FUNCTION_BLOCK CardboardCornerGuardEx EXTENDS SectionEx
VAR
	robotLeft, robotRight : REFERENCE TO Robot;
	
	insertionLeft, insertionRight : REFERENCE TO Insertion;
	insertionBottom : REFERENCE TO TeknicEIP;
	
	wrapper : REFERENCE TO WrapMachine;
	overhead : REFERENCE TO STRING;
	
	skidLeft, skidRight : REFERENCE TO MaterialStorage; //cardboard
	magazineLeft, magazineRight : REFERENCE TO MaterialStorage; //corner guard
	
	benderLeft : REFERENCE TO FoldingMachine;
END_VAR
VAR
	pushConveyorPos: REAL;
	wrapConveyorPos : REAL;
	
	insertionSlots : ARRAY[Surface.TOP_LEFT..Surface.BOTTOM_RIGHT] OF STRING;
	
	combinedCardboardCornerGuard : ARRAY[0..2*GVL.maxPairs] OF PositionMaterials;
	recipesCombined : BOOL;
	
	materialsArr : POINTER TO PositionMaterials; //array of PositionMaterials
	currentPair : REFERENCE TO PositionMaterials;
	
	frontCoverPlaced : BOOL;
	backCoverPlaced : BOOL;
	
	cornerSetLeft, cornerSetRight : INT;
	
	iWrap : INT;
	
	step : (PLACE_FRONT_COVER := -10, PLACE_BACK_COVER := -20, RUN_TO_POSITION, LOAD_FLATS, PUSH, RUN_TO_WRAP_POSITION, WRAP_AND_RELEASE, RESET);
	robotLeftOutputs, robotRightOutputs : ARRAY[1..50] OF INT;
END_VAR

entryRefPos := pushConveyorPos;
exitRefPos := wrapConveyorPos;

SUPER^();

CASE status OF
	SectionStatus.IDLE:
		RETURN;
	
	SectionStatus.ALIGNING:
		IF NOT recipesCombined THEN
			combine(
				currentBundle.cardboard, 
				currentBundle.cornerGuard, 
				combinedCardboardCornerGuard, 
				currentBundle.cardboard_over_cornerGuard);
				
			recipesCombined := TRUE;
		END_IF
		
	SectionStatus.ACTIVE:
		recipesCombined := FALSE;
		
	SectionStatus.CLEARING:
		//
		
	SectionStatus.COMPLETE:	
		//
		
	-100:
		RETURN;
		
END_CASE

METHOD changeRobotsEOAT : BOOL
VAR_INPUT
END_VAR
(*
IF robotLeft.tool <> sectionID THEN
	MEMSET(ADR(robotLeftOutputs), 0, SIZEOF(robotLeftOutputs));
	//robotLeftOutputs[1] := A21.TOOL_CHANGE_CHIPBOARD;
	robotLeft.setParamsAndWait(robotLeftOutputs);
END_IF

IF robotRight.tool <> sectionID THEN
	MEMSET(ADR(robotRightOutputs), 0, SIZEOF(robotRightOutputs));
	//robotRightOutputs[1] := A21.TOOL_CHANGE_CHIPBOARD;
	robotRight.setParamsAndWait(robotRightOutputs);
END_IF

changeRobotsEOAT := robotLeft.tool = sectionID AND robotRight.tool = sectionID;
*)
END_METHOD

METHOD PROTECTED combine : BOOL
VAR_IN_OUT
	cardboard : ARRAY[*] OF PositionMaterials;
	cornerGuard : ARRAY[*] OF PositionMaterials;
	
	combined : ARRAY[*] OF PositionMaterials;
END_VAR
VAR_INPUT
	cardboard_over_cornerGuard : BOOL;
END_VAR
VAR_INST
	topLength : REAL;
	leftLength : REAL;
	rightLength : REAL;
	bottomLength : REAL;
	
	topLeftLength : REAL;
	topRightLength : REAL;
	bottomLeftLength : REAL;
	bottomRightLength : REAL;
	
	outerMaterialLength : REAL;
	innerMaterialLength : REAL;
	
	i : INT;
	iCardboard : INT;
	iCornerGuard : INT;
END_VAR
FOR i:=0 TO GVL.maxPairs*2 BY 1 DO
	IF //no more cardboard (reached end of array or unused entries), 
		(iCardboard >= GVL.maxPairs OR_ELSE NOT PositionIsValid(cardboard[iCardboard])) AND_THEN //no more valid cardboard entries
		iCornerGuard < GVL.maxPairs AND_THEN //still has remaining corner guard
		PositionIsValid(cornerGuard[iCornerGuard]) //remaining corner guard is valid		
	THEN //finish with cornerguard
		combined[i] := cornerGuard[iCornerGuard];
		iCornerGuard := iCornerGuard + 1;
		CONTINUE;
	END_IF
	
	IF //no more cornerguard (reached end of array or unused entries)
		(iCornerGuard >= GVL.maxPairs OR_ELSE NOT PositionIsValid(cornerGuard[iCornerGuard])) AND_THEN
		iCardboard < GVL.maxPairs AND_THEN
		PositionIsValid(cardboard[iCardboard])
	THEN //finish with cardboard
		combined[i] := cardboard[iCardboard];
		iCardboard := iCardboard + 1;
		CONTINUE;
	END_IF
	
	(*
	IF NOT cardboard_over_cornerGuard THEN //cardboard on inside
		setOrder(cardboard, cornerGuard, combined, iCardboard, iCornerGuard, i);
		
	ELSE //cardboard on outside
		setOrder(cornerGuard, cardboard, combined, iCornerGuard, iCardboard, i);
		
	END_IF
	*)
END_FOR

combine := TRUE;
END_METHOD

METHOD initHardware : BOOL
conveyors := ADR(allConveyors);

robotLeft REF= robots[3];
robotRight REF= robots[4];
(*
insertionLeft REF= Hardware.insertionCardboardCornerGuardSides[Surface.LEFT];
insertionRight REF= Hardware.insertionCardboardCornerGuardSides[Surface.RIGHT];

wrapper REF= Hardware.wrapperCardboardCornerguard;
overhead REF= Hardware.overhead;

skidLeft REF= Hardware.cardboardSkid[Surface.LEFT];
skidRight REF= Hardware.cardboardSkid[Surface.RIGHT];

magazineLeft REF= Hardware.cornerGuardMagazine[Surface.LEFT];
magazineRight REF= Hardware.cornerGuardMagazine[Surface.RIGHT];

benderLeft REF= Hardware.cardboardBender[Surface.LEFT];
*)

insertionLeft REF= insertionA22Left;
insertionRight REF= insertionA22Right;

wrapper REF= wrapperA22;
overhead REF= Hardware.overhead;

skidLeft REF= cardboardSkidLeft;
skidRight REF= cardboardSkidRight;

magazineLeft REF= cornerGuardMagazineLeft;
magazineRight REF= cornerGuardMagazineRight;

benderLeft REF= cardboardBenderLeft;
END_METHOD

METHOD PROTECTED leftBendingSequence : BOOL
VAR_IN_OUT
	actingRobot : Robot;
	actingSkid : MaterialStorage;
	
	actingLoadStep : INT;
	actingRobotStep : INT;
END_VAR
VAR_INPUT
	materialID : STRING;
	foldPosition1 : INT;
	foldPosition2 : INT;
END_VAR
VAR_OUTPUT
	fail : BOOL;
END_VAR
VAR
	slot : INT;
END_VAR
END_METHOD

METHOD PROTECTED leftOverheadSequence : BOOL
VAR_IN_OUT
	actingRobot : Robot;
	actingSkid : MaterialStorage;
	
	actingLoadStep : INT;
	actingRobotStep : INT;
END_VAR
VAR_INPUT
	materialID : STRING;
	foldPosition1 : INT;
	foldPosition2 : INT;
END_VAR
VAR_OUTPUT
	fail : BOOL;
END_VAR
VAR
	slot : INT;
END_VAR
(*
CASE actingLoadStep OF
	0: //skid to bender
		IF NOT actingSkid.findSlot(materialID, position=> slot) THEN
			fail := TRUE;
			RETURN;
		END_IF
		
		IF
			actingRobot.reserve() AND_THEN
			actingRobot.setCommandAndWait(
				task:= A22.TRANSFER_TO_BENDER, 
				param0:= slot, 
				param1:= foldPosition1, 
				param2:= foldPosition2)
		THEN
			actingRobotStep := 10;
		END_IF
		
	10: //bend
		(*
		IF bendingMachine.done THEN
			cardboardCornersLoadStep := 20;
		END_IF
		*)
		
	20: //bender to overhead
		IF overhead <> '' THEN
			RETURN;
		END_IF
		
		IF
			actingRobot.reserve() AND_THEN
			actingRobot.setCommandAndWait(
				task:= A22.TRANSFER_TO_OVERHEAD, 
				param0:= 0, 
				param1:= 0, 
				param2:= 0)
		THEN
			actingRobotStep := 10;
		END_IF
		
		CASE actingRobotStep OF
			COMMAND: //send command
				IF NOT actingRobot.reserve() THEN
					RETURN;
				END_IF
				
				IF actingSkid.findSlot(currentPair.topRight, position=> slot) THEN
					actingRobot.command(
						task:= A22.TRANSFER_TO_OVERHEAD, 
						param0:= 0, 
						param1:= 0, 
						param2:= 0);
						
				ELSE
					fail := TRUE;
					RETURN;
					
				END_IF
				
			WAIT:
				IF actingRobot.done THEN
					overhead := materialID;
					
					actingRobot.release();
					actingRobotStep := 30;
					actingLoadStep := Surface.BOTTOM_RIGHT;
				END_IF
		END_CASE
END_CASE
*)
END_METHOD

METHOD PROTECTED leftRobotCornersSequence : BOOL
VAR_IN_OUT
	actingRobot : Robot;
	skid : MaterialStorage;
	loadStep : INT;
END_VAR
VAR_INPUT
	surfaceID : Surface;
	materialID : STRING;
	foldPos0 : INT;
	foldPos1 : INT;
END_VAR
VAR_OUTPUT
	fail : BOOL;
END_VAR
VAR
	slot : INT;
	
	task : INT;
	param0, param1, param2 : INT;
END_VAR
IF materialID = '' THEN
	leftRobotCornersSequence := TRUE;
	RETURN;
END_IF

IF NOT benderLeft.busy THEN
	benderLeft.foldPos0 := foldPos0;
	benderLeft.foldPos1 := foldPos1;
END_IF

CASE loadStep OF
	0: //skid to bender
		IF NOT skid.findSlot(materialID, atSlot=> slot) THEN
			fail := TRUE;
			RETURN;
		END_IF
		
		IF
			actingRobot.setCommandAndWait(
				task:= A22.TRANSFER_TO_BENDER, 
				param1:= slot, 
				param2:= foldPos0, 
				param3:= foldPos1)
		THEN
			loadStep := 10;
		END_IF
		
	10: //bend
		//IF benderLeft.done THEN
			loadStep := 20;
		//END_IF
		
		
	20: //bender to overhead or left insertion
		CASE surfaceID OF
			Surface.TOP_RIGHT, Surface.BOTTOM_RIGHT: //transfer to overhead
				IF overhead <> '' THEN
					RETURN;
				END_IF
				task := A22.TRANSFER_TO_OVERHEAD;
				
			Surface.TOP_LEFT: //load to insertion
				task:= A22.LOAD_BENDER_TO_UPPER_CORNER;
					
			Surface.BOTTOM_LEFT: //load to insertion
				task := A22.LOAD_BENDER_TO_LOWER_CORNER;
				
		END_CASE
		
		IF
			actingRobot.setCommandAndWait(
				task:= task, 
				param1:= param0, 
				param2:= param1, 
				param3:= param1)
		THEN
			 loadStep := COMPLETE;
		END_IF
	
	COMPLETE:
		//turn on suction
		leftRobotCornersSequence := TRUE;
	
END_CASE
END_METHOD

METHOD PROTECTED load : BOOL
VAR_INPUT
	pair : REFERENCE TO PositionMaterials;
END_VAR
VAR
	nextPair : REFERENCE TO PositionMaterials REF= materialsArr[iPair + 1];
	finished : BOOL;
END_VAR
(*
this method only loads corner materials (L-cardboards and corner guards)
to load flat cardboards, use loadFlats()
*)

IF NOT (robotLeft.operational AND robotRight.operational) THEN
	error := TRUE;
	currentBypass := TRUE;
	RETURN;
END_IF

IF NOT (robotLeft.reserve(sectionID) AND robotRight.reserve(sectionID)) THEN //both robots must be reserved first
	RETURN;
END_IF


IF //if next material has same position as this material, only happens if this material is cardboard and next is corner guard
	nextPair.position = pair.position AND_THEN
	NOT loadCornerGuards(nextPair, fail=> ) //load next pair (corner guards) first
THEN
	RETURN;
END_IF


IF MatchesMaterialType(pair:= pair, materialType:= 'CAR') THEN //is cardboard
	load := loadCornerCardboards(pair:= pair);

ELSIF MatchesMaterialType(pair:= pair, materialType:= 'COR') THEN //is corner guard
	load := loadCornerGuards(pair:= pair);

END_IF


IF load THEN
	robotLeft.release(sectionID);
	robotRight.release(sectionID);
END_IF
END_METHOD

METHOD PROTECTED loadBottom : BOOL
VAR_IN_OUT
	actingRobot : Robot;
	actingStorage : MaterialStorage;
	actingLoadStep : INT;
END_VAR
VAR_INPUT
	material : STRING;
END_VAR
VAR_OUTPUT
	fail : BOOL;
END_VAR
VAR
	slot : INT;
END_VAR
IF material = '' THEN
	loadBottom := TRUE;
	RETURN;
END_IF

CASE actingLoadStep OF
	0:
		IF NOT actingStorage.findSlot(materialID := material, atSlot => slot) THEN
			fail := TRUE;
			RETURN;
		END_IF
		
		IF
			actingRobot.setCommandAndWait( //perform the task
				task:= A22.LOAD_CARDBOARD_BOTTOM,
				param1:= slot,
				param2:= 0,
				param3:= 0)
		THEN
			actingLoadStep := COMPLETE;
		END_IF
		
	COMPLETE:
		//turn on suction
		loadBottom := TRUE;
	
END_CASE
END_METHOD

METHOD PROTECTED loadBottomLeft : BOOL
VAR_IN_OUT
	actingRobot : Robot;
	actingStorage : MaterialStorage;
	actingLoadStep : INT;
END_VAR
VAR_INPUT
	material : STRING;
END_VAR
VAR_OUTPUT
	fail : BOOL;
END_VAR
VAR
	slot : INT;
END_VAR
IF material = '' THEN
	loadBottomLeft := TRUE;
	RETURN;
END_IF

CASE actingLoadStep OF
	0:
		IF NOT actingStorage.findSlot(materialID := material, atSlot => slot) THEN //load from staging table
			fail := TRUE;
			RETURN;
		END_IF
		
		IF
			actingRobot.setCommandAndWait( //perform the task
				task:= A22.LOAD_CORNER_GUARD_LOWER,
				param1:= slot,
				param2:= 0,
				param3:= 0)
		THEN
			actingLoadStep := COMPLETE;
		END_IF
		
	COMPLETE:
		loadBottomLeft := TRUE;
END_CASE
END_METHOD

METHOD PROTECTED loadBottomRight : BOOL
VAR_IN_OUT
	actingRobot : Robot;
	actingStorage : MaterialStorage;
	actingLoadStep : INT;
END_VAR
VAR_INPUT
	material : STRING;
END_VAR
VAR_OUTPUT
	fail : BOOL;
END_VAR
VAR
	slot : INT;
END_VAR
IF material = '' THEN
	loadBottomRight := TRUE;
	RETURN;
END_IF

CASE actingLoadStep OF
	0:
		IF NOT actingStorage.findSlot(materialID := material, atSlot => slot) THEN //load from staging table
			fail := TRUE;
			RETURN;
		END_IF
		
		IF
			actingRobot.setCommandAndWait( //perform the task
				task:= A22.LOAD_CORNER_GUARD_LOWER,
				param1:= slot,
				param2:= 0,
				param3:= 0)
		THEN
			actingLoadStep := COMPLETE;
		END_IF
		
	COMPLETE:
		loadBottomRight := TRUE;
END_CASE
END_METHOD

METHOD PROTECTED loadCornerCardboards : BOOL
VAR_INPUT
	pair : REFERENCE TO PositionMaterials;
END_VAR
IF cornerSetLeft = 0 THEN //LEFT SIDE
	cornerSetLeft := Surface.TOP_RIGHT;
END_IF

IF
	leftRobotCornersSequence(
		actingRobot:= robotLeft, 
		skid:= skidLeft, 
		surfaceID:= cornerSetLeft,
		loadStep:= loadStepLeft, 
		materialID:= pair.topRight, 
		foldPos0:= currentBundle.cardboardFolds[cornerSetLeft][iPair],
		foldPos1:= 0,
		fail=> )
THEN
	CASE cornerSetLeft OF
		Surface.TOP_RIGHT: 
			cornerSetLeft := Surface.TOP_LEFT;
			loadStepLeft := 0;
			
		Surface.TOP_LEFT: 
			cornerSetLeft := Surface.BOTTOM_RIGHT;
			loadStepLeft := 0;
			
		Surface.BOTTOM_RIGHT: 
			cornerSetLeft := Surface.BOTTOM_LEFT;
			loadStepLeft := 0;
			
		Surface.BOTTOM_LEFT: 
			cornerSetLeft := COMPLETE;
			loadStepLeft := COMPLETE;
			
		COMPLETE:
			//
			
	END_CASE
END_IF



IF cornerSetRight = 0 THEN //RIGHT SIDE
	cornerSetRight := Surface.TOP_RIGHT;
END_IF

IF
	rightRobotCornersSequence(
		actingRobot:= robotRight, 
		skid:= skidRight, 
		loadStep:= loadStepRight, 
		materialID:= pair.topRight, 
		surfaceID:= cornerSetRight,
		foldPos1:= currentBundle.cardboardFolds[cornerSetRight][iPair], 
		foldPos2:= 0, 
		fail=> )
THEN
	CASE cornerSetRight OF
		Surface.TOP_RIGHT: 
			cornerSetRight := Surface.BOTTOM_RIGHT;
			loadStepRight := 0;
			
		Surface.BOTTOM_RIGHT: 
			cornerSetRight := COMPLETE;			
			loadStepRight := COMPLETE;
			
		COMPLETE:
			//
			
	END_CASE
END_IF


IF cornerSetLeft = COMPLETE AND cornerSetRight = COMPLETE THEN
	loadCornerCardboards := TRUE;
	
	loadStepLeft := loadStepRight := 0;
	cornerSetLeft := cornerSetRight := 0;
END_IF
END_METHOD

METHOD PROTECTED loadCornerGuards : BOOL
VAR_INPUT
	pair : REFERENCE TO PositionMaterials;
END_VAR
VAR_OUTPUT
	fail : BOOL;
END_VAR
VAR
	leftFail : BOOL;
	rightFail : BOOL;
END_VAR
CASE loadSet OF
	0: //upper corners
		IF 
			loadCornerGuardSequence(
				actingRobot:= robotLeft, 
				robotOutputs:= robotLeftOutputs, 
				actingStorage:= skidLeft, 
				actingLoadStep:= loadStepLeft, 
				surfaceID:= Surface.TOP_LEFT, 
				material:= pair.topLeft, 
				fail=> leftFail)
			AND
			loadCornerGuardSequence(
				actingRobot:= robotRight, 
				robotOutputs:= robotRightOutputs, 
				actingStorage:= skidRight,
				actingLoadStep:= loadStepRight, 
				surfaceID:= Surface.TOP_RIGHT, 
				material:= pair.topRight, 
				fail=> rightFail)
		THEN
			loadStepLeft := loadStepRight := 0;
			loadSet := 10;
		END_IF
		
	10: //lower corners
		IF 
			loadCornerGuardSequence(
				actingRobot:= robotLeft, 
				robotOutputs:= robotLeftOutputs, 
				actingStorage:= skidLeft, 
				actingLoadStep:= loadStepLeft, 
				surfaceID:= Surface.BOTTOM_LEFT, 
				material:= pair.bottomLeft, 
				fail=> leftFail)
			AND
			loadCornerGuardSequence(
				actingRobot:= robotRight, 
				robotOutputs:= robotRightOutputs, 
				actingStorage:= skidRight,
				actingLoadStep:= loadStepRight, 
				surfaceID:= Surface.BOTTOM_RIGHT, 
				material:= pair.bottomRight, 
				fail=> rightFail)
		THEN
			loadStepLeft := loadStepRight := 0;
			loadSet := COMPLETE;
		END_IF
	
	COMPLETE:
		loadStepLeft := loadStepRight := 0;
		loadSet := 0;
		
		loadCornerGuards := TRUE;
END_CASE

fail := MAX(leftFail, rightFail);
END_METHOD

METHOD loadCornerGuardSequence : BOOL
VAR_IN_OUT
	actingRobot : Robot;
	robotOutputs : ARRAY[1..50] OF INT;
	actingStorage : MaterialStorage;
	actingLoadStep : INT;
END_VAR
VAR_INPUT
	surfaceID : Surface;
	material : STRING;
END_VAR
VAR_OUTPUT
	fail : BOOL;
END_VAR
VAR
	slot : INT;
END_VAR
IF material = '' THEN
	loadCornerGuardSequence := TRUE;
	RETURN;
END_IF

CASE actingLoadStep OF
	0:
		IF NOT actingStorage.findSlot(materialID := material, atSlot => slot) THEN //load from staging table
			fail := TRUE;
			RETURN;
		END_IF
		
		MEMSET(ADR(robotOutputs), 0, SIZEOF(robotOutputs));
		CASE surfaceID OF
			Surface.TOP_LEFT, Surface.TOP_RIGHT: 		robotOutputs[1] := A22.LOAD_CORNER_GUARD_UPPER;
			Surface.BOTTOM_LEFT, Surface.BOTTOM_RIGHT:	robotOutputs[1] := A22.LOAD_CORNER_GUARD_LOWER;
		END_CASE
		robotOutputs[2] := slot;
		
		IF actingRobot.setParamsAndWait(robotOutputs) THEN
			actingLoadStep := COMPLETE;
		END_IF
		
	COMPLETE:
		//outerSuctions[surfaceID].enable := TRUE;
		loadCornerGuardSequence := TRUE;
END_CASE
END_METHOD

METHOD PROTECTED loadFlats : BOOL
VAR_INPUT
	pair : REFERENCE TO PositionMaterials;
END_VAR
CASE loadSet OF
	0: //top and bottom
		IF 
			loadTop(robotLeft, skidLeft, loadStepLeft, pair.top, fail=> ) AND
			loadBottom(robotRight, skidRight, loadStepRight, pair.bottom, fail=> )
		THEN
			loadStepLeft := loadStepRight := 0;
			loadSet := 10;
		END_IF
		
	10: //sides
		IF 
			loadSides(robotLeft, skidLeft, loadStepLeft, pair.top, fail=> ) AND
			loadSides(robotRight, skidRight, loadStepRight, pair.bottom, fail=> )
		THEN
			loadStepLeft := loadStepRight := 0;
			loadSet := COMPLETE;
		END_IF
	
	COMPLETE:
		loadStepLeft := loadStepRight := 0;
		loadSet := 0;
		
		loadFlats := TRUE;
END_CASE
END_METHOD

METHOD loadFlatSequence : BOOL
VAR_IN_OUT
	actingRobot : Robot;
	robotOutputs : ARRAY[1..50] OF INT;
	actingStorage : MaterialStorage;
	actingLoadStep : INT;
END_VAR
VAR_INPUT
	surfaceID : Surface;
	material : STRING;
END_VAR
VAR_OUTPUT
	fail : BOOL;
END_VAR
VAR
	slot : INT;
END_VAR
IF material = '' THEN
	loadFlatSequence := TRUE;
	RETURN;
END_IF

CASE actingLoadStep OF
	0:
		IF NOT actingStorage.findSlot(materialID := material, atSlot => slot) THEN
			fail := TRUE;
			RETURN;
		END_IF
		
		MEMSET(ADR(robotOutputs), 0, SIZEOF(robotOutputs));
		CASE surfaceID OF
			Surface.TOP: 					robotOutputs[1] := A22.LOAD_CARDBOARD_TOP;
			Surface.LEFT, Surface.RIGHT: 	robotOutputs[1] := A22.LOAD_CARDBOARD_SIDE;
			Surface.BOTTOM: 				robotOutputs[1] := A22.LOAD_CARDBOARD_BOTTOM;
		END_CASE
		robotOutputs[2] := slot;
		
		IF actingRobot.setParamsAndWait(robotOutputs) THEN
			actingLoadStep := COMPLETE;
		END_IF
		
	COMPLETE:
		loadFlatSequence := TRUE;
	
END_CASE
END_METHOD

METHOD PROTECTED loadSides : BOOL
VAR_IN_OUT
	actingRobot : Robot;
	actingStorage : MaterialStorage;
	actingLoadStep : INT;
END_VAR
VAR_INPUT
	material : STRING;
END_VAR
VAR_OUTPUT
	fail : BOOL;
END_VAR
VAR
	slot : INT;
END_VAR
IF material = '' THEN
	loadSides := TRUE;
	RETURN;
END_IF

CASE actingLoadStep OF
	0:
		IF NOT actingStorage.findSlot(materialID := material, atSlot => slot) THEN
			fail := TRUE;
			RETURN;
		END_IF
		
		IF
			actingRobot.setCommandAndWait( //perform the task
				task:= A22.LOAD_CARDBOARD_SIDE,
				param1:= slot,
				param2:= 0,
				param3:= 0)
		THEN
			actingLoadStep := COMPLETE;
		END_IF
		
	COMPLETE:
		//turn suction on
		loadSides := TRUE;
END_CASE
END_METHOD

METHOD PROTECTED loadTop : BOOL
VAR_IN_OUT
	actingRobot : Robot;
	actingStorage : MaterialStorage;
	actingLoadStep : INT;
END_VAR
VAR_INPUT
	material : STRING;
END_VAR
VAR_OUTPUT
	fail : BOOL;
END_VAR
VAR
	slot : INT;
END_VAR
IF material = '' THEN
	loadTop := TRUE;
	RETURN;
END_IF

CASE actingLoadStep OF
	0:
		IF NOT actingStorage.findSlot(materialID := material, atSlot => slot) THEN //load from staging table
			fail := TRUE;
			RETURN;
		END_IF
		
		IF
			actingRobot.setCommandAndWait( //perform the task
				task:= A22.LOAD_CARDBOARD_TOP,
				param1:= slot,
				param2:= 0,
				param3:= 0)
		THEN
			actingLoadStep := COMPLETE;
		END_IF
		
	COMPLETE:
		loadTop := TRUE;
END_CASE
END_METHOD

METHOD PROTECTED loadTopLeft : BOOL
VAR_IN_OUT
	actingRobot : Robot;
	actingStorage : MaterialStorage;
	actingLoadStep : INT;
END_VAR
VAR_INPUT
	material : STRING;
END_VAR
VAR_OUTPUT
	fail : BOOL;
END_VAR
VAR
	slot : INT;
END_VAR
IF material = '' THEN
	loadTopLeft := TRUE;
	RETURN;
END_IF

CASE actingLoadStep OF
	0:
		IF NOT actingStorage.findSlot(materialID := material, atSlot => slot) THEN //load from staging table
			fail := TRUE;
			RETURN;
		END_IF
		
		IF
			actingRobot.setCommandAndWait( //perform the task
				task:= A22.LOAD_CORNER_GUARD_UPPER,
				param1:= slot,
				param2:= 0,
				param3:= 0)
		THEN
			actingLoadStep := COMPLETE;
		END_IF
		
	COMPLETE:
		loadTopLeft := TRUE;
END_CASE
END_METHOD

METHOD PROTECTED loadTopRight : BOOL
VAR_IN_OUT
	actingRobot : Robot;
	actingStorage : MaterialStorage;
	actingLoadStep : INT;
END_VAR
VAR_INPUT
	material : STRING;
END_VAR
VAR_OUTPUT
	fail : BOOL;
END_VAR
VAR
	slot : INT;
END_VAR
IF material = '' THEN
	loadTopRight := TRUE;
	RETURN;
END_IF

CASE actingLoadStep OF
	0:
		IF NOT actingStorage.findSlot(materialID := material, atSlot => slot) THEN //load from staging table
			fail := TRUE;
			RETURN;
		END_IF
		
		IF
			actingRobot.setCommandAndWait( //perform the task
				task:= A22.LOAD_CORNER_GUARD_UPPER,
				param1:= slot,
				param2:= 0,
				param3:= 0)
		THEN
			actingLoadStep := COMPLETE;
		END_IF
		
	COMPLETE:
		loadTopRight := TRUE;
END_CASE
END_METHOD

METHOD placeFrontCover : BOOL
VAR_INPUT
END_VAR
END_METHOD

METHOD PROTECTED process : BOOL
VAR
	masterLength : REAL;
	targetPos : REAL;
	targetStep : INT;
END_VAR
VAR
	maxHeight : REAL := 1000; //1000mm, 100cm, 1m tall at home pos
END_VAR
(*
VAR_INST
	resumePosition : REAL;
END_VAR
VAR CONSTANT
	wrapDelta : REAL := 5;
END_VAR
*)
//TODO: write instructions for wrapping front and back covers

IF NOT frontCoverPlaced THEN
	targetPos := 0;
	
ELSIF iPair < GVL.maxPairs THEN
	targetPos := currentPair.position;
	
ELSIF NOT backCoverPlaced AND iPair >= GVL.maxPairs THEN
	targetPos := currentBundle.length;
	
ELSIF iPair >= GVL.maxPairs THEN
	process := TRUE;
	RETURN;
	
END_IF

CASE step OF
	PLACE_FRONT_COVER:
		IF placeFrontCover() THEN
			step := RUN_TO_POSITION;
		END_IF
	
	RUN_TO_POSITION:
		IF //only load corners, flats will be PUSHed when bundle arrives at position
			directionCheckAndSet(pushConveyorPos, currentPair.position) AND 
			load(pair:= currentPair)
		THEN
			step := 10;
		END_IF
		
	LOAD_FLATS:
		IF loadFlats(pair:= currentPair) THEN
			step := PUSH;
		END_IF
		
	PUSH:
		setConveyorMode(ConveyorMode.STOP);
		(*
		IF
			NOT insertionLeft.align(targetPos:= maxHeight - currentBundle.height) OR
			NOT insertionRight.align(targetPos:= maxHeight - currentBundle.height)
		THEN
			RETURN;
		END_IF
		
		insertionLeft.press();
		insertionRight.press();
		*)
		
		IF NOT insertionLeft.contact THEN
			//insertionRight.slideOut();
			insertionLeft.traverse(direction:= MC_Negative_Direction);
			insertionLeft.press();
		END_IF
		
		IF NOT insertionRight.contact THEN
			//insertionRight.slideOut();
			insertionRight.traverse(direction:= MC_Negative_Direction);
			insertionRight.press();
		END_IF
		
		(*
		IF NOT insertionBottom.contact THEN
			insertionBottom.traverse(direction := FALSE);
		END_IF
		*)
		
		IF insertionLeft.contact AND insertionRight.contact (*AND insertionBottom.contact*) THEN		
			step := RUN_TO_WRAP_POSITION;
		END_IF
		
	RUN_TO_WRAP_POSITION:
		masterLength := GetPositionMasterLength(currentPair);
		IF iWrap >= currentPair.wrapPoints THEN
			step := COMPLETE;
			RETURN;
		END_IF
		
		IF //compare current position with wrap position
			directionCheckAndSet(
				wrapConveyorPos,
				(currentPair.position - masterLength/2) + (masterLength/(currentPair.wrapPoints + 1) * (iWrap + 1)))
		THEN
			step := WRAP_AND_RELEASE;
		END_IF
		
	WRAP_AND_RELEASE: //wrap
		setConveyorMode(ConveyorMode.STOP);
		IF wrapper.ready OR (NOT wrapper.busy AND NOT wrapper.error) THEN
			wrapper.wrap(currentPair.wrapRotations);
		END_IF
		
		IF NOT insertionLeft.home THEN
			insertionLeft.align(0);
			insertionLeft.release();
		END_IF
		
		IF NOT insertionRight.home THEN
			insertionRight.align(0);
			insertionRight.release();
		END_IF
		
		IF wrapper.done AND insertionLeft.home AND insertionRight.home (*AND insertionBottom.home*) THEN
			step := WRAP_AND_RELEASE;
		END_IF
		
	COMPLETE: //reset
		setConveyorMode(ConveyorMode.FORWARD);
		
		iPair := iPair + 1;
		IF iPair >= GVL.maxPairs THEN
			iPair := 0;
			process := TRUE;
		END_IF
		iWrap := 0;
		
		step := 0;
END_CASE
END_METHOD

METHOD PROTECTED rightRobotCornersSequence : BOOL
VAR_IN_OUT
	actingRobot : Robot;
	skid : MaterialStorage;
	loadStep : INT;
END_VAR
VAR_INPUT
	surfaceID : Surface;
	materialID : STRING;
	foldPos1 : INT;
	foldPos2 : INT;
END_VAR
VAR_OUTPUT
	fail : BOOL;
END_VAR
VAR
	slot : INT;
	
	task : INT;
	param0, param1, param2 : INT;
END_VAR
IF materialID = '' THEN
	rightRobotCornersSequence := TRUE;
	RETURN;
END_IF

CASE loadStep OF
	0: //overhead to insertion
		IF overhead = '' THEN
			RETURN;
		END_IF
		
		CASE surfaceID OF
			Surface.TOP_RIGHT:
				task := A22.LOAD_OVERHEAD_TO_UPPER_CORNER;
				
			Surface.BOTTOM_RIGHT:
				task := A22.LOAD_OVERHEAD_TO_LOWER_CORNER;
				
		END_CASE
		
		IF
			actingRobot.setCommandAndWait(
				task:= task, 
				param1:= slot, 
				param2:= foldPos1, 
				param3:= foldPos2)
		THEN
			loadStep := COMPLETE;
		END_IF
	
	COMPLETE:
		//turn on suction
		rightRobotCornersSequence := TRUE;
	
END_CASE
END_METHOD

METHOD PROTECTED robotsFailed : BOOL
VAR_INPUT
END_VAR
IF NOT robotLeft.operational OR NOT robotLeft.operational THEN
	error := TRUE;
	currentBypass := TRUE;
	robotsFailed := TRUE;
END_IF
END_METHOD

METHOD PROTECTED setOrder : BOOL
VAR_IN_OUT
	innerArray : ARRAY[*] OF PositionMaterials;
	outerArray : ARRAY[*] OF PositionMaterials;
	
	combined : ARRAY[*] OF PositionMaterials;
	
	i_inner : INT;
	i_outer : INT;
	i_combined : INT;
END_VAR
VAR
	topLength : REAL;
	leftLength : REAL;
	rightLength : REAL;
	bottomLength : REAL;
	
	topLeftLength : REAL;
	topRightLength : REAL;
	bottomLeftLength : REAL;
	bottomRightLength : REAL;
	
	outerMaterialLength : REAL;
	innerMaterialLength : REAL;
END_VAR
//if inner material is in front of outer material, inner material goes first
IF innerArray[i_inner].position <= outerArray[i_outer].position THEN

	combined[i_combined] := innerArray[i_inner];
	i_inner := i_inner + 1; //check next cardboard during next iteration
	
	setOrder := TRUE;
	RETURN;
END_IF
	
outerMaterialLength := GetPositionMasterLength(outerArray[i_outer]);
innerMaterialLength := GetPositionMasterLength(innerArray[i_inner]);

//if current inner material is too close to current outer material, place inner material first
//compare inner materials' front with outer material's back
IF (innerArray[i_inner].position - innerMaterialLength/2) < (outerArray[i_outer].position + outerMaterialLength/2) THEN
	combined[i_combined] := innerArray[i_inner];
	i_inner := i_inner + 1;
ELSE //otherwise, outer material can go
	combined[i_combined] := outerArray[i_outer];
	i_outer := i_outer + 1;
END_IF

setOrder := TRUE;
END_METHOD

METHOD PROTECTED usesProcess : BOOL
VAR
	i : INT;
END_VAR
IF materialsArr = 0 THEN
	RETURN;
END_IF

FOR i:=0 TO GVL.maxPairs BY 1 DO
	IF PositionIsValid(materialsArr[i]) THEN
		usesProcess := TRUE;
		RETURN;		
	END_IF
END_FOR
END_METHOD

END_FUNCTION_BLOCK

(* stored: Version 1.1.0.1, ProductVersion 3.1.4024.11
   POU CardboardCornerGuardEx: Id {a8c59fad-2bb5-4d17-87d2-8ffaf74c5994}, SpecialFunc None
   Folder Covers: Id {7c3844f1-0007-4c8a-b6ea-281eb812ff3f}
   Folder Loading: Id {21d5f6d1-557c-44cc-9d02-c168d792f248}
   Folder Cardboard (Corner): Id {8f34b24f-0f93-4965-8f66-af279f368ca3}
   Folder Cardboard (Flat): Id {c27b3a4c-1195-4283-a5df-d05ab3293d66}
   Folder Corner Guard: Id {6556ca3f-09cb-4649-92bd-22bd27f604cb}
   Folder Recipe Combination: Id {e84711e1-12c7-48bc-a0fc-ee5336e88119}
   Folder z_Obsolete: Id {7b969d6a-6d5e-4d8d-a765-9d3f6701131b}
   Folder Special: Id {af4676bc-89a7-4b8c-af36-e757826d91f3}
   Method changeRobotsEOAT: Id {ad257d74-55b5-4856-b29b-eabb6aa02516}
   Method combine: Id {68c0a6ae-b842-4781-b6e7-e5f46d476b9d}
   Method initHardware: Id {e451f7ee-82f1-43b8-8539-8a18f14c4dc6}
   Method leftBendingSequence: Id {a327e208-1928-4adc-9c68-993330ffc2d3}
   Method leftOverheadSequence: Id {d4f60085-e53a-48fb-8343-4cf41c518967}
   Method leftRobotCornersSequence: Id {08bffef9-e349-4b7d-9ae3-92f5a7d8876a}
   Method load: Id {a681c93d-e590-4020-9185-d7ae010cf638}
   Method loadBottom: Id {96fe8dec-7975-47d9-bf27-7665a4b63d8b}
   Method loadBottomLeft: Id {ab1e7458-9ffe-4f54-b3b2-5672f3fb4d32}
   Method loadBottomRight: Id {2f89862d-4e9e-4b8f-9d60-93e8bfb6d8cd}
   Method loadCornerCardboards: Id {fc6e26f1-7233-42c4-a94a-66d2e256266a}
   Method loadCornerGuards: Id {73216583-3bb4-409e-896a-e96f29db7009}
   Method loadCornerGuardSequence: Id {6d84fe42-26e5-4a1f-b580-8cefdfabe586}
   Method loadFlats: Id {b9a93d4c-938b-4af6-a5a3-5141d50c48d4}
   Method loadFlatSequence: Id {e9b25173-0158-437d-9616-4153dd5d3500}
   Method loadSides: Id {bce6adc5-bd14-4a01-8baf-9e8ced2a7029}
   Method loadTop: Id {d3181a38-c048-40f0-a727-904bc3296946}
   Method loadTopLeft: Id {da9b7d7b-fe35-4a3e-b66b-564cfda3ebe6}
   Method loadTopRight: Id {0864a9ae-8557-457e-92f9-25a9eda0d9aa}
   Method placeFrontCover: Id {25c41d77-9114-4bb4-b025-8fd9cd529867}
   Method process: Id {10741552-30dc-43f4-b22b-a667441db858}
   Method rightRobotCornersSequence: Id {879cd7f3-c4e8-4979-a4c5-8a1bacb14790}
   Method robotsFailed: Id {0924391b-eda8-40a3-92e3-ade088e653b4}
   Method setOrder: Id {e2776e5b-59eb-47e7-a6d5-4049b002d6f5}
   Method usesProcess: Id {197330ac-793e-4729-9655-d4ff2caf3be4} *)
